# EPICS StreamDevice protocol: ip/ipApp/Db/JenaNV40.proto
# Protocol file for Piezosystems Jena NV 40/1 CLE
# http://www.piezojena.com/en/site/piezo-controller-and-amplifier__183/

############  SVN Repository information  #############
# $Date: 2011-09-28 16:47:03 -0500 (Wed, 28 Sep 2011) $
# $Author: kpetersn $
# $Revision: 13794 $
# $HeadURL: https://subversion.xray.aps.anl.gov/synApps/ip/tags/R2-15/ipApp/Db/JenaNV40.proto $
# $Id: JenaNV40.proto 13794 2011-09-28 21:47:03Z kpetersn $
#######################################################

OutTerminator = CR;
InTerminator = CR LF;

writeValue {
  out "wr,%f";
}

readValue {
  out "rd";
  in "rd,%f";
}

closedLoop {
  out "%{ol|cl}";
}

remoteControl {
  out "%{i0|i1}";
}
